% RSLogix 500 project fault_handler.RSS, saved by version 8.30.00.16 %
PROJECT "UNTITLED"    % processor: Bul.1763 MicroLogix 1100 Series B %

PROGRAM FILES
  LAD 2 "MAIN"  4 rungs
  LAD 10 "HANDLFAULT"  13 rungs

DATA FILES
  O0 OUTPUT  4 elements
  I1 INPUT  6 elements
  S2 STATUS  66 elements
  B3 BINARY  1 elements
  T4 TIMER  1 elements
  C5 COUNTER  1 elements
  R6 CONTROL  1 elements
  N7 INTEGER  10 elements
  F8 FLOAT  1 elements
  N100 ERR_LSB_CT  256 elements
  N101 ERR_MSB_CT  256 elements

LADDER 2 "MAIN"
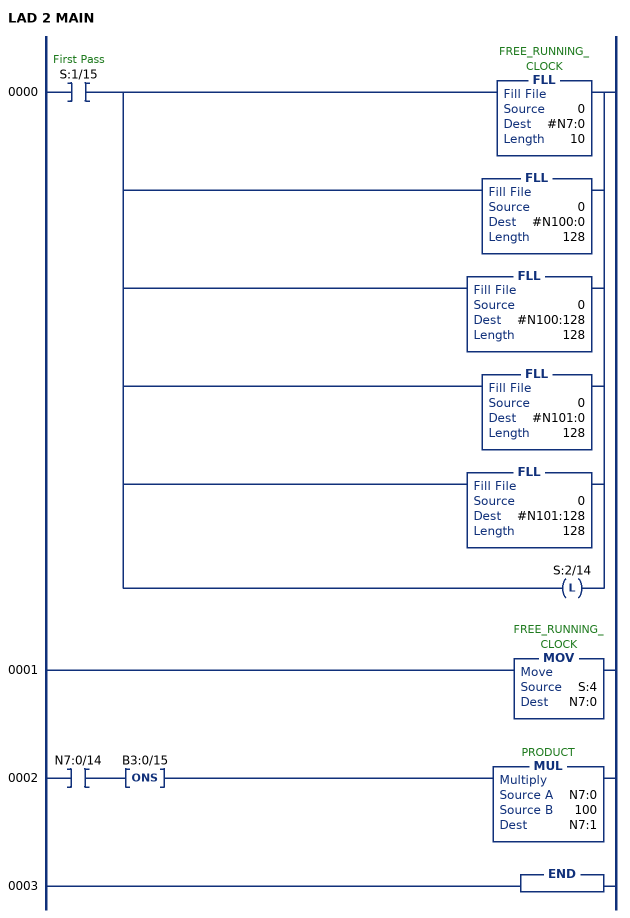
% Rung: 0 %
SOR XIC S:1/15 BST FLL 0 #N7:0 10 NXB FLL 0 #N100:0 128 NXB FLL 0 #N100:128 128 NXB FLL 0 #N101:0 128 NXB FLL 0 #N101:128 128 NXB OTL S:2/14 BND EOR
%   S:1/15  "First Pass" %
%   N7:0  FREE_RUNNING_CLOCK %
% Rung: 1 %
SOR MOV S:4 N7:0 EOR
%   S:4  "Time Base" %
%   N7:0  FREE_RUNNING_CLOCK %
% Rung: 2 %
SOR XIC N7:0/14 ONS B3:0/15 MUL N7:0 100 N7:1 EOR
%   N7:0  FREE_RUNNING_CLOCK %
%   N7:1  PRODUCT %
% Rung: 3 %
SOR END EOR

LADDER 10 "HANDLFAULT"
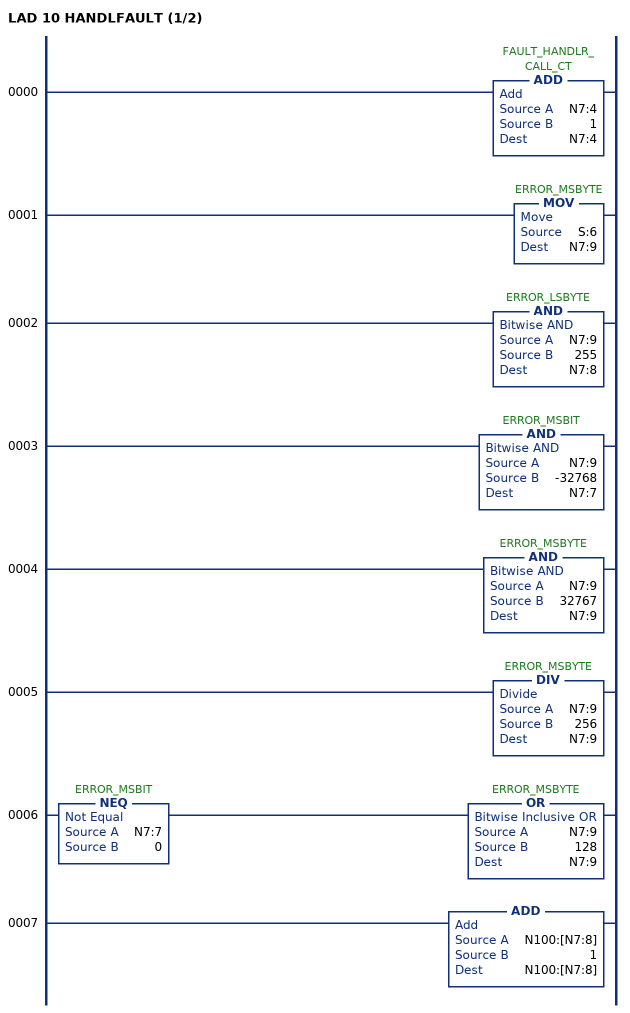
% Rung: 0 %
SOR ADD N7:4 1 N7:4 EOR
%   N7:4  FAULT_HANDLR_CALL_CT %
% Rung: 1 %
SOR MOV S:6 N7:9 EOR
%   S:6  "Major Error Fault Code" %
%   N7:9  ERROR_MSBYTE %
% Rung: 2 %
SOR AND N7:9 255 N7:8 EOR
%   N7:9  ERROR_MSBYTE %
%   N7:8  ERROR_LSBYTE %
% Rung: 3 %
SOR AND N7:9 -32768 N7:7 EOR
%   N7:9  ERROR_MSBYTE %
%   N7:7  ERROR_MSBIT %
% Rung: 4 %
SOR AND N7:9 32767 N7:9 EOR
%   N7:9  ERROR_MSBYTE %
% Rung: 5 %
SOR DIV N7:9 256 N7:9 EOR
%   N7:9  ERROR_MSBYTE %
% Rung: 6 %
SOR NEQ N7:7 0 OR N7:9 128 N7:9 EOR
%   N7:7  ERROR_MSBIT %
%   N7:9  ERROR_MSBYTE %
% Rung: 7 %
SOR ADD N100:[N7:8] 1 N100:[N7:8] EOR
%   N7:8  ERROR_LSBYTE %

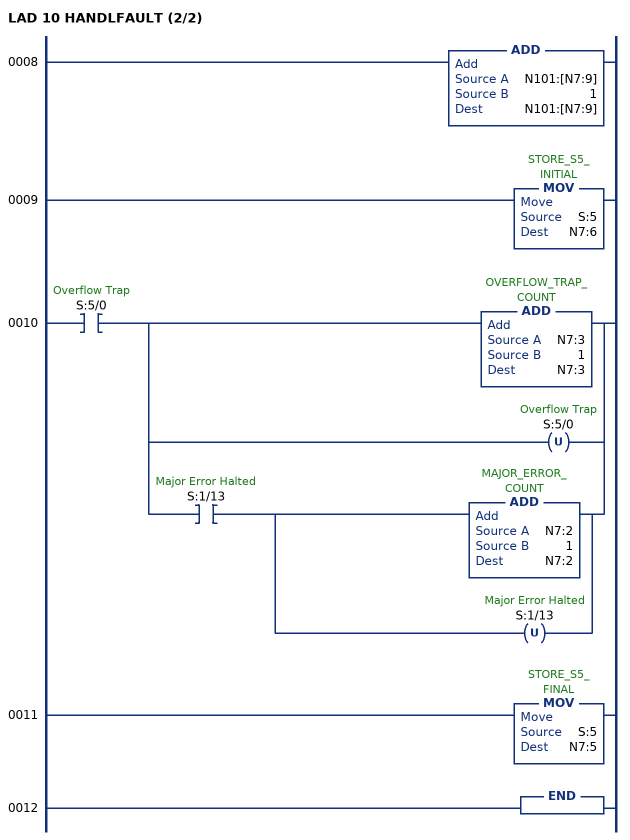
% Rung: 8 %
SOR ADD N101:[N7:9] 1 N101:[N7:9] EOR
%   N7:9  ERROR_MSBYTE %
% Rung: 9 %
SOR MOV S:5 N7:6 EOR
%   N7:6  STORE_S5_INITIAL %
% Rung: 10 %
SOR XIC S:5/0 BST ADD N7:3 1 N7:3 NXB OTU S:5/0 NXB XIC S:1/13 BST ADD N7:2 1 N7:2 NXB OTU S:1/13 BND BND EOR
%   S:5/0  "Overflow Trap" %
%   N7:3  OVERFLOW_TRAP_COUNT %
%   S:1/13  "Major Error Halted" %
%   N7:2  MAJOR_ERROR_COUNT %
% Rung: 11 %
SOR MOV S:5 N7:5 EOR
%   N7:5  STORE_S5_FINAL %
% Rung: 12 %
SOR END EOR

OTHER DOCUMENTED ADDRESSES
  8000F  

DATA TABLE (non-zero values as saved)
DATA N101
% N101:0 % 1 0 0 0 0 0 0 0 0 0
